// TwinCAT 3 PLC project Nepionic_Log
// Title: Nepionic_Log
// Company: Nepionic
// Author: Nepionic
// ProjectVersion: 0.1.1
// ProgramVersion: 3.1.4026.21
// libraries:
//   Tc2_Standard, * (Beckhoff Automation GmbH)
//   Tc2_System, * (Beckhoff Automation GmbH)
//   Tc2_Utilities, * (Beckhoff Automation GmbH)
//   Tc3_DynamicMemory, * (Beckhoff Automation GmbH)
// project tree:
//   Lib/Appenders/AdsLog/ AdsLogAppender.TcPOU, LogLevelToAdsLogMsgType.TcPOU (not stored)
//   Lib/Appenders/File/ DeleteFilesState.TcDUT (not stored), DeleteOldFiles.TcPOU (not stored), GenerateTimeData.TcPOU, GetFileAgeInSeconds.TcPOU (not stored), LoggingConfiguration.TcDUT (not stored), PersistToFileState.TcDUT (not stored), RollingIntervals.TcDUT (not stored)
//   Lib/Appenders/ LogAppender.TcIO
//   Lib/ Constants.TcGVL (not stored), DateTime.TcPOU, Error.TcDUT, ErrorCodes.TcDUT (not stored)
//   Lib/Core/ LogAttribute.TcDUT, LogAttributeType.TcDUT, LogAttributeValueToString.TcPOU (not stored), LogLevel.TcDUT
//   Lib/Manager/ GetLogManager.TcPOU, LogManager.TcPOU (not stored)
//   Lib/Logger/ DefaultLogger.TcPOU, Logger.TcIO
//   Lib/String/ AnyToString.TcPOU (not stored), DefaultStringBuilder.TcPOU, DynamicStringBuffer.TcPOU (not stored), LimitedStringBuilder.TcIO (not stored), StringBuilder.TcIO

// ---- Lib/Core/LogAttribute.TcDUT
// A single structured log attribute — a key/value pair attached to a log entry.
// Used by LogCore.LogWithAttributes and consumed by OtelLogCore.
TYPE LogAttribute :
STRUCT
	// Attribute name  e.g. 'event.name', 'previous_state'
	key : STRING(31);
	// Attribute value e.g. 'axis.state_changed', 'Idle'
	value : STRING(63);
END_STRUCT
END_TYPE

// ---- Lib/Core/LogAttributeType.TcDUT
{attribute 'qualified_only'}
{attribute 'strict'}
{attribute 'to_string'}
TYPE LogAttributeType :
(
	Uint8 := 0,
	Uint16 := 1,
	Uint32 := 2,
	Uint64 := 3,
	Int8 := 4,
	Int16 := 5,
	Int32 := 6,
	Int64 := 7,
	Boolean := 8,
	Float32 := 9,
	Float64 := 10,
	Str := 11
) USINT;
END_TYPE

// ---- Lib/Core/LogLevel.TcDUT
{attribute 'qualified_only'}
{attribute 'strict'}
{attribute 'to_string'}
TYPE LogLevel :
(
	Debug := 0,
	Information,
	Warning,
	Error,
	Fatal
);
END_TYPE

// ---- Lib/Error.TcDUT
/// This is the error type used in this library.
TYPE Error :
STRUCT
  /// `TRUE` signals an active error
	Active : BOOL;
  /// Error code of type `ErrorCodes`
	Code : INT;
  /// Plain text error message
	Info : Tc2_System.T_MaxString;
END_STRUCT
END_TYPE

// ---- Lib/Appenders/LogAppender.TcIO
/// Sink interface implemented by every log appender.
/// `LogManager` fans log records out to each registered appender whose `Level`
/// threshold is satisfied.
///
/// Implementations must be silent — logging infrastructure must never fault
/// application code, so `Append` should never raise an exception or leave
/// an error that the caller must handle.
INTERFACE PUBLIC LogAppender EXTENDS __System.IQueryInterface

/// Deliver one log record to this appender.
/// Called by `LogManager.Dispatch` for every record whose level meets the
/// appender's `Level` threshold.
METHOD PUBLIC Append : BOOL
VAR_INPUT
	/// Severity of the log record.
	level : LogLevel;
	/// Free-text log message.
	message : Tc2_System.T_MaxString;
	/// Structured source identifier (instance path or logger name).
	source : Tc2_System.T_MaxString;
	/// Structured key/value attributes attached to this record.
	attributes : ARRAY[0..9] OF LogAttribute;
	/// Number of populated entries in `attrs` (0 – 10).
	attribute_count : USINT;
END_VAR
END_METHOD

/// Minimum severity this appender accepts.
/// Records whose level is strictly below this threshold are silently dropped
/// by `LogManager` before `Append` is ever called.
{attribute 'monitoring' := 'call'}
PROPERTY PUBLIC Level : LogLevel
GET
END_GET
SET
END_SET
END_PROPERTY

END_INTERFACE

// ---- Lib/Logger/Logger.TcIO
/// User-facing logging interface.
/// Implemented by `DefaultLogger` and any test doubles.
///
/// For structured attributes use the concrete `DefaultLogger` type directly,
/// which adds `WithAttribute` and `OnCondition` chaining methods.
INTERFACE PUBLIC Logger EXTENDS __System.IQueryInterface

/// Log at DEBUG level.
METHOD PUBLIC Debug : BOOL
VAR_INPUT
	message : Tc2_System.T_MaxString;
END_VAR
END_METHOD

/// Log at ERROR level.
METHOD PUBLIC Error : BOOL
VAR_INPUT
	message : Tc2_System.T_MaxString;
END_VAR
END_METHOD

/// Log at FATAL level.
METHOD PUBLIC Fatal : BOOL
VAR_INPUT
	message : Tc2_System.T_MaxString;
END_VAR
END_METHOD

/// Log at INFORMATION level.
METHOD PUBLIC Info : BOOL
VAR_INPUT
	message : Tc2_System.T_MaxString;
END_VAR
END_METHOD

/// Log at WARNING level.
METHOD PUBLIC Warning : BOOL
VAR_INPUT
	message : Tc2_System.T_MaxString;
END_VAR
END_METHOD

END_INTERFACE

// ---- Lib/String/StringBuilder.TcIO
{attribute 'hide'}
INTERFACE INTERNAL StringBuilder

METHOD Append : StringBuilder // Append text TO t current build STRING.
VAR_INPUT
    Text : Tc2_System.T_MaxString; //Text to append to current build string
END_VAR
END_METHOD

METHOD AppendIf : StringBuilder
VAR_INPUT
    Condition : BOOL;
    Text : Tc2_System.T_MaxString;
END_VAR
END_METHOD

METHOD InsertAtLocation : StringBuilder
VAR_INPUT
    Text : Tc2_System.T_MaxString;
    Position : INT;
END_VAR
END_METHOD

METHOD PadLeft : StringBuilder
VAR_INPUT
    text : Tc2_System.T_MaxString; // Text to append to current build string
    length : INT; // Total length of text + padding
    c : STRING(1); // Character to be padded left of text
END_VAR
END_METHOD

METHOD Reset : LimitedStringBuilder //Reset current build STRING TO an empty STRING.
END_METHOD

METHOD ToString : Tc2_System.T_MaxString //Returns current build STRING.
END_METHOD

END_INTERFACE

// ---- Lib/Appenders/AdsLog/AdsLogAppender.TcPOU
/// Log appender that writes to the TwinCAT ADS output window via `AdsLogStr`.
///
/// Register once at startup:
/// ```st
/// GetLogManager().Register(ads_appender);
/// ```
///
/// Optional: raise the threshold above DEBUG to reduce output noise:
/// ```st
/// ads_appender.Level := LogLevel.Warning;
/// ```
{attribute 'linkalways'}
{attribute 'no_explicit_call' := 'This FB is a CLASS and must be accessed using methods or properties'}
{attribute 'enable_dynamic_creation'}
FUNCTION_BLOCK PUBLIC AdsLogAppender IMPLEMENTS LogAppender
VAR
	_level : LogLevel := LogLevel.Debug;
END_VAR

METHOD Append : BOOL
VAR_INPUT
	level : LogLevel;
	message : Tc2_System.T_MaxString;
	source : Tc2_System.T_MaxString;
	attributes : ARRAY[0..9] OF LogAttribute;
	attribute_count : USINT;
END_VAR
VAR
	msg_type : DWORD;
	text : Tc2_System.T_MaxString;
	i : USINT;
	pair : Tc2_System.T_MaxString;
END_VAR
msg_type := Tc2_System.AdsLog_MsgType_Log OR LogLevelToAdsLogMsgType(level);

// Build: "[source] message  {key=value, ...}"
IF Tc2_Standard.Len(source) > 0 THEN
	text := Tc2_Standard.Concat('[', Tc2_Standard.Concat(source, '] '));
END_IF
text := Tc2_Standard.Concat(text, message);

IF attribute_count > 0 THEN
	text := Tc2_Standard.Concat(text, '  {');
	FOR i := 0 TO attribute_count - 1 DO
		IF i > 0 THEN
			text := Tc2_Standard.Concat(text, ', ');
		END_IF
		pair := Tc2_Standard.Concat(attributes[i].key, Tc2_Standard.Concat('=', attributes[i].value));
		text := Tc2_Standard.Concat(text, pair);
	END_FOR
	text := Tc2_Standard.Concat(text, '}');
END_IF

Tc2_System.AdsLogStr(msg_type, text, '');
Append := TRUE;
END_METHOD

{attribute 'monitoring' := 'call'}
PROPERTY Level : LogLevel
GET
Level := _level;
END_GET
SET
_level := Level;
END_SET
END_PROPERTY

END_FUNCTION_BLOCK

// ---- Lib/Appenders/File/GenerateTimeData.TcPOU
FUNCTION_BLOCK GenerateTimeData
VAR_OUTPUT
	timeAsFileTime : Tc2_Utilities.T_FILETIME;
	timeAsSystemTime : Tc2_Utilities.TIMESTRUCT;
	timeAsString : Tc2_System.T_MaxString;
	utcTimeAsFileTime : Tc2_Utilities.T_FILETIME;
END_VAR
VAR
	_localSystemTime : Tc2_Utilities.FB_LocalSystemTime;
	_getSystemTime : Tc2_System.GETSYSTEMTIME;
	_timeZoneInfo : Tc2_Utilities.FB_GetTimeZoneInformation;
	_localTime : Tc2_Utilities.FB_SystemTimeToTzSpecificLocalTime;
	_localSystemTimeValid : Tc2_Standard.R_TRIG;
	_utcTime : Tc2_Utilities.FB_TzSpecificLocalTimeToFileTime;
END_VAR
VAR_TEMP
	utcSystemTime : Tc2_Utilities.TIMESTRUCT;
END_VAR

_localSystemTime(
	sNetID	:=	'',
	bEnable := 	TRUE,
	dwCycle	:=	1,
	dwOpt	:=	1,
	tTimeout:=	DEFAULT_ADS_TIMEOUT
);

_timeZoneInfo(
	sNetID := '',
	bExecute := TRUE,
	tTimeout := DEFAULT_ADS_TIMEOUT);

_UtcTime(
	in := SYSTEMTIME_TO_FILETIME(timeAsSystemTime),
	tzInfo := _timeZoneInfo.tzInfo);
	
timeAsSystemTime 	:=	_localSystemTime.systemTime;
timeAsFileTime 		:= 	SYSTEMTIME_TO_FILETIME(timeAsSystemTime);
timeAsString 		:= 	SYSTEMTIME_TO_STRING(timeAsSystemTime);
utcTimeAsFileTime	:= 	_utcTime.out;

_localSystemTimeValid(CLK := _localSystemTime.bValid);

{attribute 'monitoring':='call'}
PROPERTY Done : BOOL
GET
Done := _localSystemTimeValid.Q;
END_GET
END_PROPERTY

// Replaces placeholders in format string by the actual time values
METHOD PRIVATE ReplaceFormatPlaceholder : STRING
VAR_INPUT
	Format : STRING;
	Length : INT;
	TimeType : STRING(1);
END_VAR
VAR_INST
	i : INT;
	replaceString : STRING;
	timeString : STRING;
END_VAR
IF    TimeType = 'Y' 	THEN timeString := TO_STRING(timeAsSystemTime.wYear); 
ELSIF TimeType = 'M' 	THEN timeString := TO_STRING(timeAsSystemTime.wMonth); 
ELSIF TimeType = 'D' 	THEN timeString := TO_STRING(timeAsSystemTime.wDay); 
ELSIF TimeType = 'h' 	THEN timeString := TO_STRING(timeAsSystemTime.wHour); 
ELSIF TimeType = 'm' 	THEN timeString := TO_STRING(timeAsSystemTime.wMinute); 
ELSIF TimeType = 's' 	THEN timeString := TO_STRING(timeAsSystemTime.wSecond); 
ELSIF TimeType = 'i' 	THEN timeString := TO_STRING(timeAsSystemTime.wMilliseconds); 
ELSE
  timeString:='';
END_IF

replaceString := '';

IF Length > LEN(timeString) THEN
	FOR i:=1 TO Length - LEN(timeString) DO
		replaceString := Tc2_Standard.CONCAT(replaceString, '0');
	END_FOR
	replaceString := Tc2_Standard.CONCAT(replaceString, timeString);
ELSE
	replaceString := RIGHT(timeString, Length);
END_IF

ReplaceFormatPlaceholder := REPLACE(Format, replaceString, Length, FIND(Format, TimeType));
END_METHOD

// Returns a formatted string containing the actual time information 
//	Y : year
//	M : month
// 	D : day
//  h : hour 
//  m : minute
//  s : second
//  i : millisecond
// 
// Example: _YYMMDD-hh:mm:ss:iii_
// => _20210812-12:30:22:123_
METHOD ToString : Tc2_System.T_MaxString
VAR_INPUT
	Format : STRING;
END_VAR
VAR_INST
	inputString : STRING;
	char : STRING(1);
	formattedString : Tc2_System.T_MaxString;
END_VAR
VAR
	year : INT := 0;
	month : INT := 0;
	day : INT := 0;
	hour : INT := 0;
	minute : INT := 0;
	second : INT := 0;
	millisecond : INT := 0;
END_VAR
VAR CONSTANT
	VALID_FORMAT : STRING := 'YMDhms';
END_VAR
// Parses "Format" and returns a adequatly formatted string containing the time information
inputString := Format;

WHILE LEN(inputString) > 0 DO
	char := LEFT(inputString, 1);
	
	IF    char = 'Y' THEN 	year := year + 1;
	ELSIF char = 'M' THEN	month := month + 1;
	ELSIF char = 'D' THEN	day := day + 1;
	ELSIF char = 'h' THEN	hour := hour + 1;
	ELSIF char = 'm' THEN	minute := minute + 1;
	ELSIF char = 's' THEN 	second := second + 1;
	ELSIF char = 'i' THEN 	millisecond := millisecond + 1;
	END_IF
	
	inputString := DELETE(inputString, 1, 1);
END_WHILE

formattedString := ReplaceFormatPlaceholder(Format, year, 'Y');
formattedString := ReplaceFormatPlaceholder(formattedString, month, 'M');
formattedString := ReplaceFormatPlaceholder(formattedString, day, 'D');
formattedString := ReplaceFormatPlaceholder(formattedString, hour, 'h');
formattedString := ReplaceFormatPlaceholder(formattedString, minute, 'm');
formattedString := ReplaceFormatPlaceholder(formattedString, second, 's');
formattedString := ReplaceFormatPlaceholder(formattedString, millisecond, 'i');

ToString := formattedString;
END_METHOD

END_FUNCTION_BLOCK

// ---- Lib/DateTime.TcPOU
/// Generate time data in different formats.
{attribute: 'hide_all_locals'}
FUNCTION_BLOCK PUBLIC DateTime
VAR
	local_system_time : Tc2_Utilities.Fb_LocalSystemTime;
	get_system_time : Tc2_System.GetSystemTime;
	time_zone_info : Tc2_Utilities.Fb_GetTimeZoneInformation;
	local_Time : Tc2_Utilities.Fb_SystemTimeToTzSpecificLocalTime;
	local_system_time_valid : Tc2_Standard.R_Trig;
	utc_time : Tc2_Utilities.Fb_TzSpecificLocalTimeToFileTime;
END_VAR

// Get local system time
local_system_time(
	sNetID  :=  '',
	bEnable :=  TRUE,
	dwCycle :=  1,
	dwOpt :=  1,
	tTimeout:= Tc2_System.Default_Ads_Timeout
);

// Get timezone information
time_zone_info(
	sNetID := '',
	bExecute := TRUE,
	tTimeout := Tc2_System.Default_Ads_Timeout
);

// Convert local time to utc time
utc_time(
	in := THIS^.AsLocalFileTime,
	tzInfo := time_zone_info.tzInfo
);
  
// Finished retrieving time data
local_system_time_valid(Clk := local_system_time.bValid);

/// Returns local time as `Tc2_Utilities.T_FILETIME`.
{attribute 'monitoring':='variable'}
PROPERTY AsLocalFileTime : Tc2_Utilities.T_FILETIME
GET
AsLocalFileTime := Tc2_Utilities.SystemTime_To_FileTime(THIS^.AsLocalSystemTime);
END_GET
END_PROPERTY

/// Returns local time as `Tc2_Utilities.TIMESTRUCT`.
{attribute 'monitoring':='variable'}
PROPERTY AsLocalSystemTime : Tc2_Utilities.TIMESTRUCT
GET
AsLocalSystemTime := local_system_time.systemTime;
END_GET
END_PROPERTY

/// Returns local time as string.
{attribute 'monitoring':='variable'}
PROPERTY AsLocalSystemTimeString : Tc2_System.T_MAXSTRING
GET
AsLocalSystemTimeString := Tc2_Utilities.SYSTEMTIME_TO_STRING(THIS^.AsLocalSystemTime);
END_GET
END_PROPERTY

/// Returns UTC time as `Tc2_Utilities.T_FILETIME`.
{attribute 'monitoring':='variable'}
PROPERTY AsUtcFileTime : Tc2_Utilities.T_FILETIME
GET
AsUtcFileTime := utc_time.out;
END_GET
END_PROPERTY

/// When calling `DateTime` the first time, it takes some time until all time and timezone information is available.
/// `Done` is `TRUE` for one cycle, once all the data is ready. 
{attribute 'monitoring':='call'}
PROPERTY Done : BOOL
GET
Done := local_system_time_valid.Q;
END_GET
END_PROPERTY

// Replaces placeholders in format string by the actual time values.
{attribute 'hide_all_locals'}
{attribute 'hide'}
METHOD PRIVATE ReplaceFormatPlaceholder : STRING
VAR_INPUT
	format : STRING;
	length : INT;
	time_type : STRING(1);
END_VAR
VAR_INST
	i : INT;
	replace_string : STRING;
	time_string : STRING;
END_VAR
VAR
	local_system_time : Tc2_Utilities.TimeStruct;
END_VAR
local_system_time := THIS^.AsLocalSystemTime;

IF    time_type = 'Y'  THEN time_string := TO_STRING(local_system_time.wYear); 
ELSIF time_type = 'M'  THEN time_string := TO_STRING(local_system_time.wMonth); 
ELSIF time_type = 'D'  THEN time_string := TO_STRING(local_system_time.wDay); 
ELSIF time_type = 'h'  THEN time_string := TO_STRING(local_system_time.wHour); 
ELSIF time_type = 'm'  THEN time_string := TO_STRING(local_system_time.wMinute); 
ELSIF time_type = 's'  THEN time_string := TO_STRING(local_system_time.wSecond); 
ELSIF time_type = 'i'  THEN time_string := TO_STRING(local_system_time.wMilliseconds); 
ELSE
  time_string:='';
END_IF

replace_string := '';

IF length > Tc2_Standard.Len(time_string) THEN
	FOR i:=1 TO length - Tc2_Standard.Len(time_string) DO
		replace_string := Tc2_Standard.ConCat(replace_string, '0');
	END_FOR
	replace_string := Tc2_Standard.ConCat(replace_string, time_string);
ELSE
	replace_string := Tc2_Standard.Right(time_string, length);
END_IF

ReplaceFormatPlaceholder := Tc2_Standard.Replace(format, replace_string, length, Tc2_Standard.Find(format, time_type));
END_METHOD

/// Returns a formatted string containing the actual time information 
/// - `Y` : year
/// - `M` : month
/// - `D` : day
/// - `h` : hour 
/// - `m` : minute
/// - `s` : second
/// - `i` : millisecond
/// 
/// Example:    
/// _YYMMDD-hh:mm:ss:iii_   
/// => _20210812-12:30:22:123_
{attribute 'hide_all_locals'}
METHOD ToFormatString : Tc2_System.T_MaxString
VAR_INPUT
  /// Format the timestamp should have.
  format : STRING;
END_VAR
VAR_INST
  inputString : STRING;
  c : STRING(1);
  formattedString : Tc2_System.T_MaxString;
END_VAR
VAR
  year : INT := 0;
  month : INT := 0;
  day : INT := 0;
  hour : INT := 0;
  minute : INT := 0;
  second : INT := 0;
  millisecond : INT := 0;
END_VAR
VAR CONSTANT
  ValidFormat : STRING := 'YMDhms';
END_VAR
// Parses "format" and returns a adequatly formatted string containing the time information
inputString := format;

WHILE Tc2_Standard.LEN(inputString) > 0 DO
  c := Tc2_Standard.LEFT(inputString, 1);
  
  IF    c = 'Y' THEN year := year + 1;
  ELSIF c = 'M' THEN month := month + 1;
  ELSIF c = 'D' THEN day := day + 1;
  ELSIF c = 'h' THEN hour := hour + 1;
  ELSIF c = 'm' THEN minute := minute + 1;
  ELSIF c = 's' THEN second := second + 1;
  ELSIF c = 'i' THEN millisecond := millisecond + 1;
  END_IF
  
  inputString := Tc2_Standard.DELETE(inputString, 1, 1);
END_WHILE

formattedString := ReplaceFormatPlaceholder(format, year, 'Y');
formattedString := ReplaceFormatPlaceholder(formattedString, month, 'M');
formattedString := ReplaceFormatPlaceholder(formattedString, day, 'D');
formattedString := ReplaceFormatPlaceholder(formattedString, hour, 'h');
formattedString := ReplaceFormatPlaceholder(formattedString, minute, 'm');
formattedString := ReplaceFormatPlaceholder(formattedString, second, 's');
formattedString := ReplaceFormatPlaceholder(formattedString, millisecond, 'i');

ToFormatString := formattedString;
END_METHOD

END_FUNCTION_BLOCK

// ---- Lib/Manager/GetLogManager.TcPOU
/// Returns a reference to the process-global `LogManager` singleton.
///
/// The singleton is a `VAR_STAT` inside this FUNCTION — no GVL required.
///
/// Usage:
/// ```st
/// // Register an appender at startup:
/// GetLogManager().Register(my_otel_appender);
///
/// // Raise the global floor to Information:
/// GetLogManager().Level := LogLevel.Information;
/// ```
FUNCTION PUBLIC GetLogManager : REFERENCE TO LogManager
VAR_STAT
	_instance : LogManager;
END_VAR

GetLogManager REF= _instance;

END_FUNCTION

// ---- Lib/Logger/DefaultLogger.TcPOU
/// Concrete logger that dispatches to the process-global `LogManager` singleton.
///
/// Declare one instance per component/axis/subsystem and pass `name` to
/// `FB_Init` — the name becomes the `source` field on every log record so
/// you can filter by component in your log viewer.
///
/// Simple usage:
/// ```st
/// VAR
///   log : DefaultLogger('AxisX');
/// END_VAR
/// log.Info('Homing started');
/// log.Error('Limit switch triggered');
/// ```
///
/// Structured attributes and conditional logging:
/// ```st
/// log.WithAttribute('state', 'Homing').WithAttribute('speed', '100').Info('Axis moving');
/// log.OnCondition(error_active).Error('Drive fault detected');
/// ```
///
/// No wiring required — `FB_Init` connects automatically to `GetLogManager()`.
/// Register appenders on `GetLogManager()` once at program startup.
{attribute 'linkalways'}
{attribute 'no_explicit_call' := 'This FB is a CLASS and must be accessed using methods or properties'}
{attribute 'enable_dynamic_creation'}
FUNCTION_BLOCK PUBLIC DefaultLogger IMPLEMENTS Logger
VAR
	_name : STRING(63);
	attributes : ARRAY[0..9] OF LogAttribute;
	attribute_count : USINT;
	condition : BOOL := TRUE;
	chain_started : BOOL;
END_VAR

/// Log at DEBUG level.
METHOD PUBLIC Debug : BOOL
VAR_INPUT
	message : Tc2_System.T_MaxString;
END_VAR
InitChain();
IF condition THEN
	GetLogManager().Dispatch(LogLevel.Debug, message, _name, attributes, attribute_count);
END_IF
ResetChain();
Debug := TRUE;
END_METHOD

/// Log at ERROR level.
METHOD PUBLIC Error : BOOL
VAR_INPUT
	message : Tc2_System.T_MaxString;
END_VAR
InitChain();
IF condition THEN
	GetLogManager().Dispatch(LogLevel.Error, message, _name, attributes, attribute_count);
END_IF
ResetChain();
Error := TRUE;
END_METHOD

/// Log at FATAL level.
METHOD PUBLIC Fatal : BOOL
VAR_INPUT
	message : Tc2_System.T_MaxString;
END_VAR
InitChain();
IF condition THEN
	GetLogManager().Dispatch(LogLevel.Fatal, message, _name, attributes, attribute_count);
END_IF
ResetChain();
Fatal := TRUE;
END_METHOD

METHOD FB_Init : BOOL
VAR_INPUT
	bInitRetains : BOOL;
	bInCopyCode  : BOOL;
	/// Component name used as the `source` field on every log record.
	name : STRING(63);
END_VAR
_name := name;
END_METHOD

/// Log at INFORMATION level.
METHOD PUBLIC Info : BOOL
VAR_INPUT
	message : Tc2_System.T_MaxString;
END_VAR
InitChain();
IF condition THEN
	GetLogManager().Dispatch(LogLevel.Information, message, _name, attributes, attribute_count);
END_IF
ResetChain();
Info := TRUE;
END_METHOD

// Initialise chain state on the first call of a log chain.
// Idempotent — safe to call from every chain method.
{attribute 'hide'}
METHOD PRIVATE InitChain
IF NOT chain_started THEN
	chain_started := TRUE;
	condition := TRUE;
	attribute_count := 0;
END_IF
END_METHOD

/// Component name used as the `source` field on every log record.
{attribute 'monitoring' := 'call'}
PROPERTY PUBLIC Name : STRING(63)
GET // PUBLIC
Name := _name;
END_GET
SET // PUBLIC
_name := Name;
END_SET
END_PROPERTY

/// Conditionally emit the log record.
/// When `cond` is FALSE the chain is still initialised but the terminal
/// method (`Debug`, `Info`, etc.) will be a no-op.
/// ```st
/// log.OnCondition(error_active).Error('Drive fault');
/// ```
METHOD PUBLIC OnCondition : REFERENCE TO DefaultLogger
VAR_INPUT
	cond : BOOL;
END_VAR
InitChain();
condition := cond;
OnCondition REF= THIS^;
END_METHOD

// Reset chain state after a terminal method completes.
// Must be called at the end of every Debug/Info/Warning/Error/Fatal implementation.
{attribute 'hide'}
METHOD PRIVATE ResetChain
chain_started := FALSE;
condition := TRUE;
attribute_count := 0;
END_METHOD

/// Log at WARNING level.
METHOD PUBLIC Warning : BOOL
VAR_INPUT
	message : Tc2_System.T_MaxString;
END_VAR
InitChain();
IF condition THEN
	GetLogManager().Dispatch(LogLevel.Warning, message, _name, attributes, attribute_count);
END_IF
ResetChain();
Warning := TRUE;
END_METHOD

/// Attach a structured key/value attribute to the current log record.
/// Call before the terminal method (`Debug`, `Info`, `Warning`, `Error`, `Fatal`).
/// Up to 10 attributes per record; extras are silently ignored.
/// This method is chainable:
/// ```st
/// log.WithAttribute('key1', 'val1').WithAttribute('key2', 'val2').Info('msg');
/// ```
METHOD PUBLIC WithAttribute : REFERENCE TO DefaultLogger
VAR_INPUT
	key : STRING(31);
	value : STRING(63);
END_VAR
InitChain();

IF attribute_count < 10 THEN
	attributes[attribute_count].key   := key;
	attributes[attribute_count].value := value;
	attribute_count := attribute_count + 1;
END_IF

WithAttribute REF= THIS^;
END_METHOD

END_FUNCTION_BLOCK

// ---- Lib/String/DefaultStringBuilder.TcPOU
FUNCTION_BLOCK INTERNAL DefaultStringBuilder IMPLEMENTS StringBuilder, LimitedStringBuilder
VAR
	{attribute 'hide'}
	work_string : Tc2_System.T_MaxString;
END_VAR

METHOD PUBLIC Append : StringBuilder // Append text TO t current build STRING.
VAR_INPUT
	text : Tc2_System.T_MaxString; //text to append to current build string
END_VAR
work_string := Tc2_Standard.Concat(work_string, text);
Append := THIS^;
END_METHOD

METHOD PUBLIC AppendIf : StringBuilder
VAR_INPUT
	condition : BOOL;
	text : Tc2_System.T_MaxString;
END_VAR
IF condition THEN
	work_string := Tc2_Standard.Concat(work_string, text);
END_IF
AppendIf := THIS^;
END_METHOD

METHOD PUBLIC InsertAtLocation : StringBuilder
VAR_INPUT
	text : Tc2_System.T_MaxString;
	position : INT;
END_VAR
work_string := Tc2_Standard.Insert(work_string, text, position);
InsertAtLocation  := THIS^;
END_METHOD

METHOD PadLeft : StringBuilder
VAR_INPUT
	text : Tc2_System.T_MaxString; // Text to append to current build string
	length : INT; // Total length of text + padding
	c : STRING(1); // Character to be padded left of text
END_VAR
VAR
	i : INT;
	pad_length : INT;
END_VAR
// Add left padding
pad_length := Tc2_Standard.Len(text) - length;
FOR i := 1 TO pad_length DO
	work_string:= Tc2_Standard.Concat(work_string, c);
END_FOR

// Add text
work_string:= Tc2_Standard.Concat(work_string, text);

PadLeft := THIS^;
END_METHOD

METHOD PUBLIC Reset : LimitedStringBuilder //Reset current build STRING TO an empty STRING.
work_string := '';
Reset := THIS^;
END_METHOD

METHOD PUBLIC ToString : Tc2_System.T_MaxString //Returns current build STRING.
ToString := work_string;
END_METHOD

END_FUNCTION_BLOCK
